FUNCTION CONVERT_MASS_TO_FLOW : REAL
VAR_INPUT
	Mass:REAL; (*in gramme*)
	Delay:TIME; (*in ms*)
END_VAR
VAR
END_VAR

CONVERT_MASS_TO_FLOW:=Mass/TIME_TO_DWORD(Delay)*60000;

END_FUNCTION

(* stored: Version 1.1.0.1, ProductVersion 3.1.0.26
   POU CONVERT_MASS_TO_FLOW: Id {a63d694c-a9df-481c-9da5-a534eed52d1b} *)
